FUNCTION_BLOCK FB_SituarPale_SFC

VAR_IN_OUT
	  TpoPaleEntrada: TIME;
END_VAR

VAR_INPUT
    // SFC-Flags
    SFCPause: BOOL;
    SFCReset: BOOL;
    
    // Indicadores de sincronizacion
    Ack: BOOL := TRUE;
    Execute: BOOL;
    
    // Entradas
    PresenciaPale: BOOL;
    CodigoPaleBit0: BOOL;
    CodigoPaleBit1: BOOL;
    CodigoPaleBit2: BOOL;    
END_VAR
VAR_OUTPUT
    // Indicadores de sincronizacion
    Done: BOOL;
    Ready: BOOL;
    
    // Parametros
    CodigoPale: BYTE;
    
    // Salidas
    CintaActiva: BOOL;
END_VAR
VAR
END_VAR

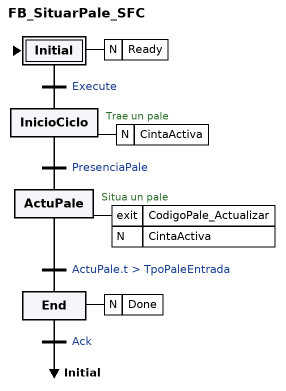
INITIAL_STEP Initial:
    Ready(N);
END_STEP
TRANSITION FROM Initial TO InicioCiclo
    := Execute;
END_TRANSITION
// Trae un pale
STEP InicioCiclo:
    CintaActiva(N);
END_STEP
TRANSITION FROM InicioCiclo TO ActuPale
    := PresenciaPale;
END_TRANSITION
// Situa un pale
STEP ActuPale:
    CodigoPale_Actualizar(P0);  // exit action
    CintaActiva(N);
END_STEP
TRANSITION FROM ActuPale TO End
    := ActuPale.t > TpoPaleEntrada;
END_TRANSITION
STEP End:
    Done(N);
END_STEP
TRANSITION FROM End TO Initial
    := Ack;
END_TRANSITION

ACTION CodigoPale_Actualizar:
CodigoPale.0 := CodigoPaleBit0;
CodigoPale.1 := CodigoPaleBit1;
CodigoPale.2 := CodigoPaleBit2;
END_ACTION

END_FUNCTION_BLOCK

(* stored: Version 1.1.0.1, ProductVersion 3.1.4024.9
   POU FB_SituarPale_SFC: Id {874a499f-85d8-470a-bd97-def0802233cc}, SpecialFunc None
   Action CodigoPale_Actualizar: Id {1a4d1bfd-f666-4c8c-9f54-d5f78029b7dd} *)
